FUNCTION_BLOCK FB_System_AFA_600
VAR_INPUT
	Freigabe_auto								: BOOL;
	Freigabe_Deakt_auto							: BOOL;
	Betrieb_Anford_auto							: BOOL;
	Regelung_Modus_auto							: SINT;
	Regelung_Sollw_auto							: REAL;
END_VAR
VAR_OUTPUT
	{attribute 'OPC.UA.DA' := '1'}Steuerung				: ST_System_AFA_Steuerung;		
	{attribute 'OPC.UA.DA' := '1'}Stellwert				: ST_System_AFA_Stellwert;		
	{attribute 'OPC.UA.DA' := '1'}Zustand					: ST_System_AFA_Zustand;	
	{attribute 'OPC.UA.DA' := '1'}Parameter				: ST_System_AFA_Parameter;		
END_VAR
VAR
	Pumpe_600				: FB_PU;
	Pumpe_235				: FB_PU;
	Pumpe_690				: FB_PU_Schuetz;
	Stellventil_605			: FB_SVs;
	Stellventil_235			: FB_SVs;
	Regelventil_600			: FB_RV;
	Regelventil_Ost_640		: FB_RV;
	Regelventil_West_660	: FB_RV;

	Zustandscheck			: FB_System_AFA_Zustandscheck;
	Logik					: FB_System_AFA_Logik;
	Ablaufsteuerung			: FB_System_AFA_Ablaufsteuerung;
	Sollwertscheck			: FB_System_AFA_Sollwertscheck;
	Regelung				: FB_System_AFA_Regelung;
	Stellwertscheck			: FB_System_AFA_Stellwertscheck;
	T_zyklus_ON: TON;
	T_zyklus_OFF: TON;


END_VAR
VAR // added by the converter: edge detectors and wires of the graphical bodies
    _w1 : BOOL;
    _w2 : ANY;
END_VAR

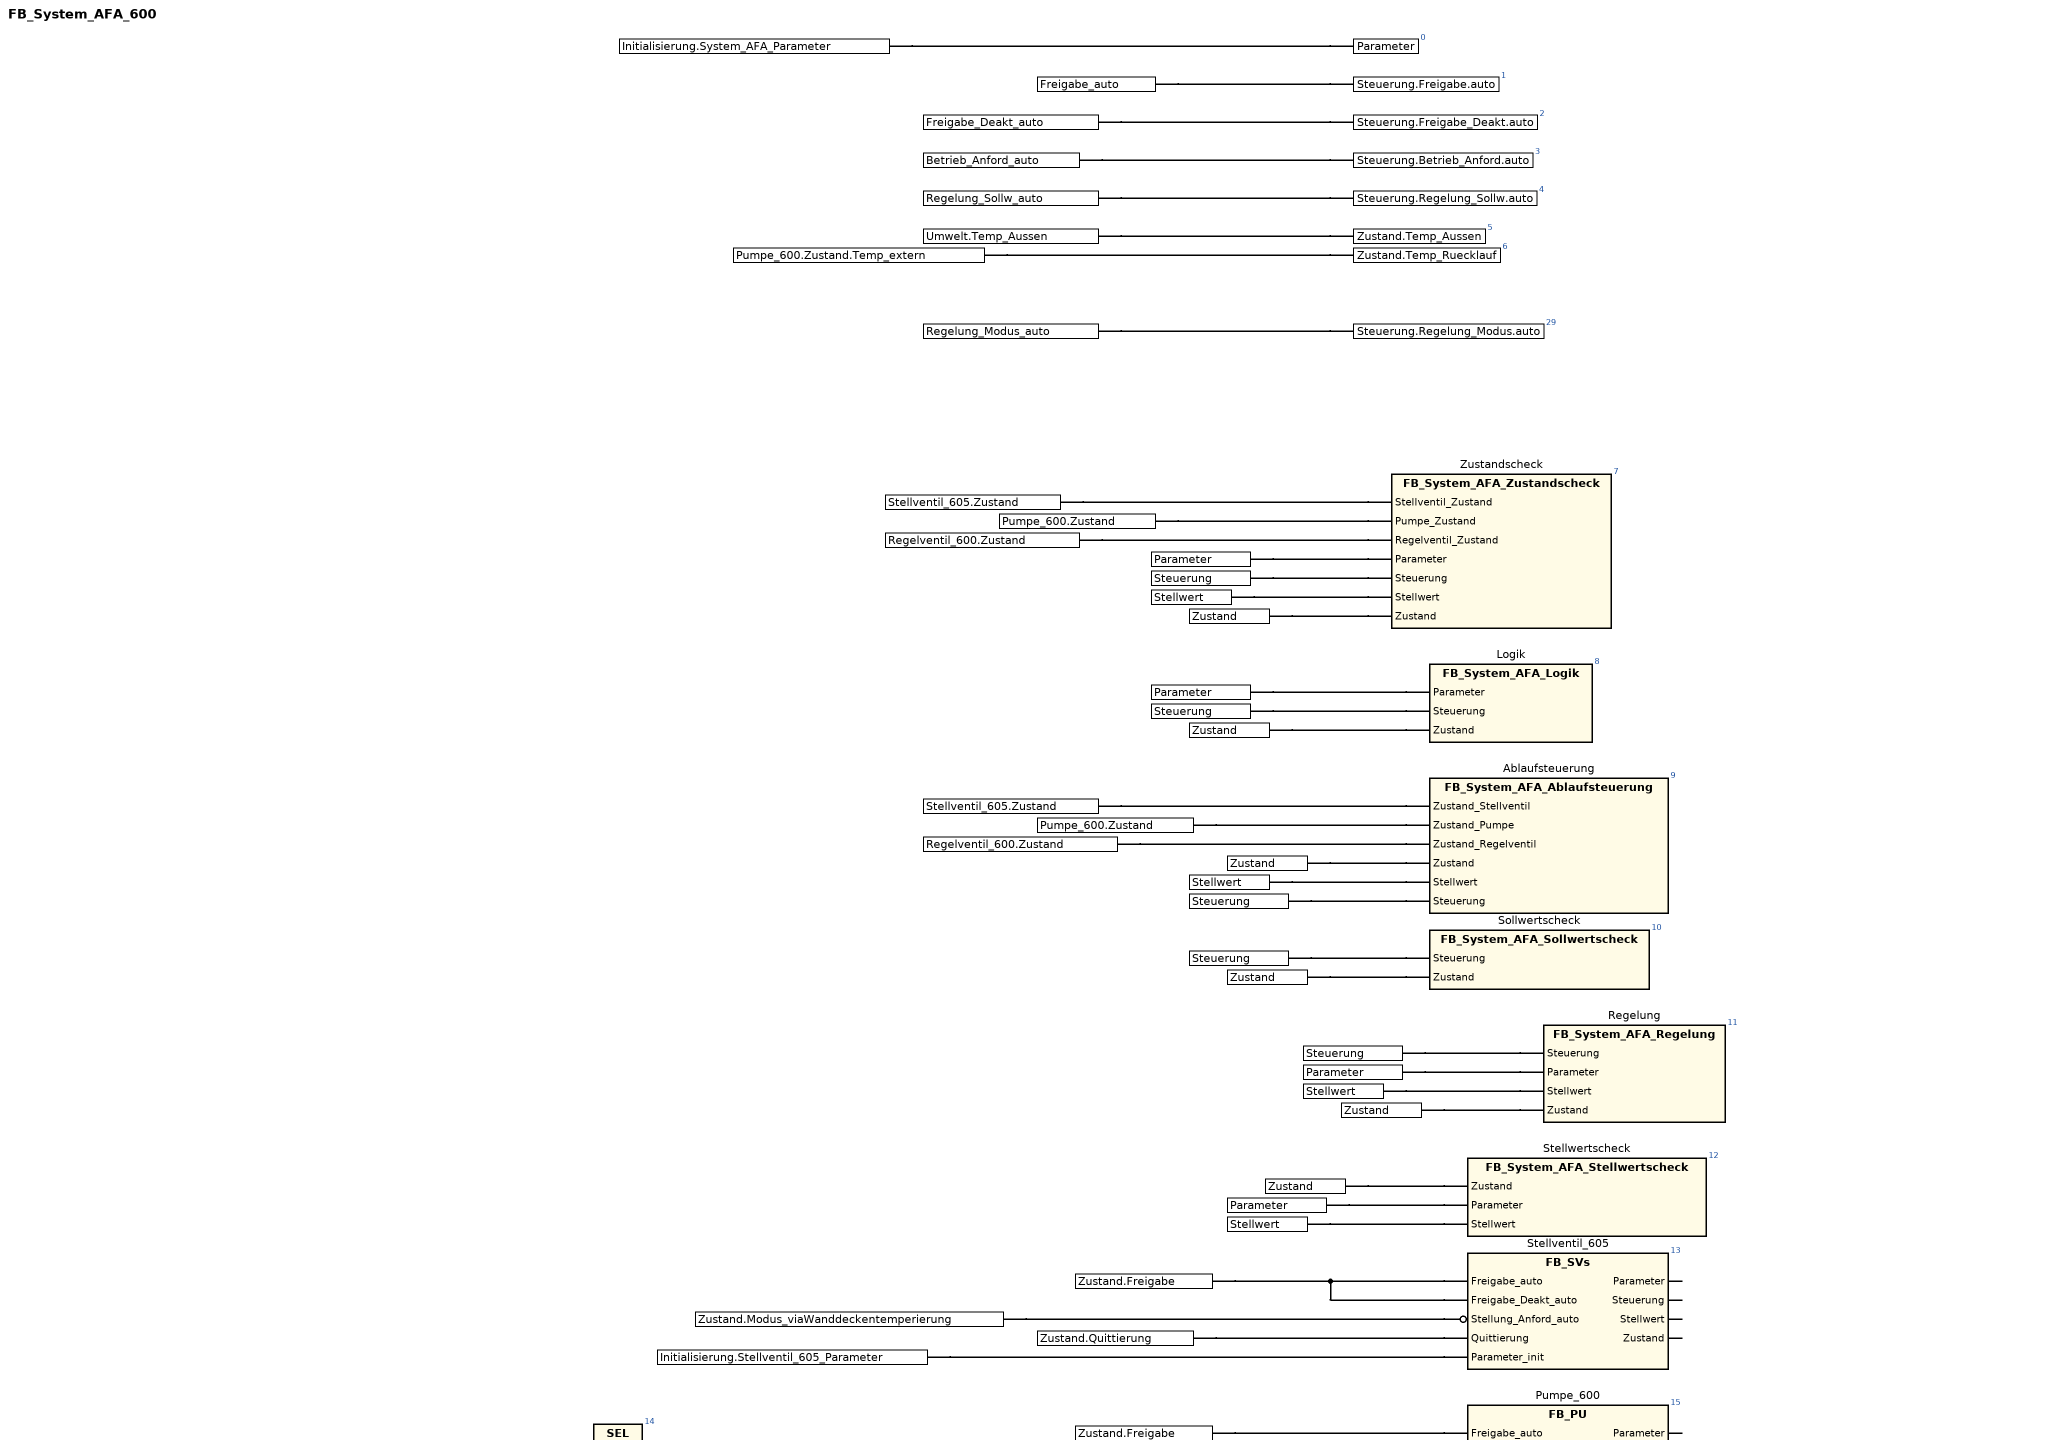
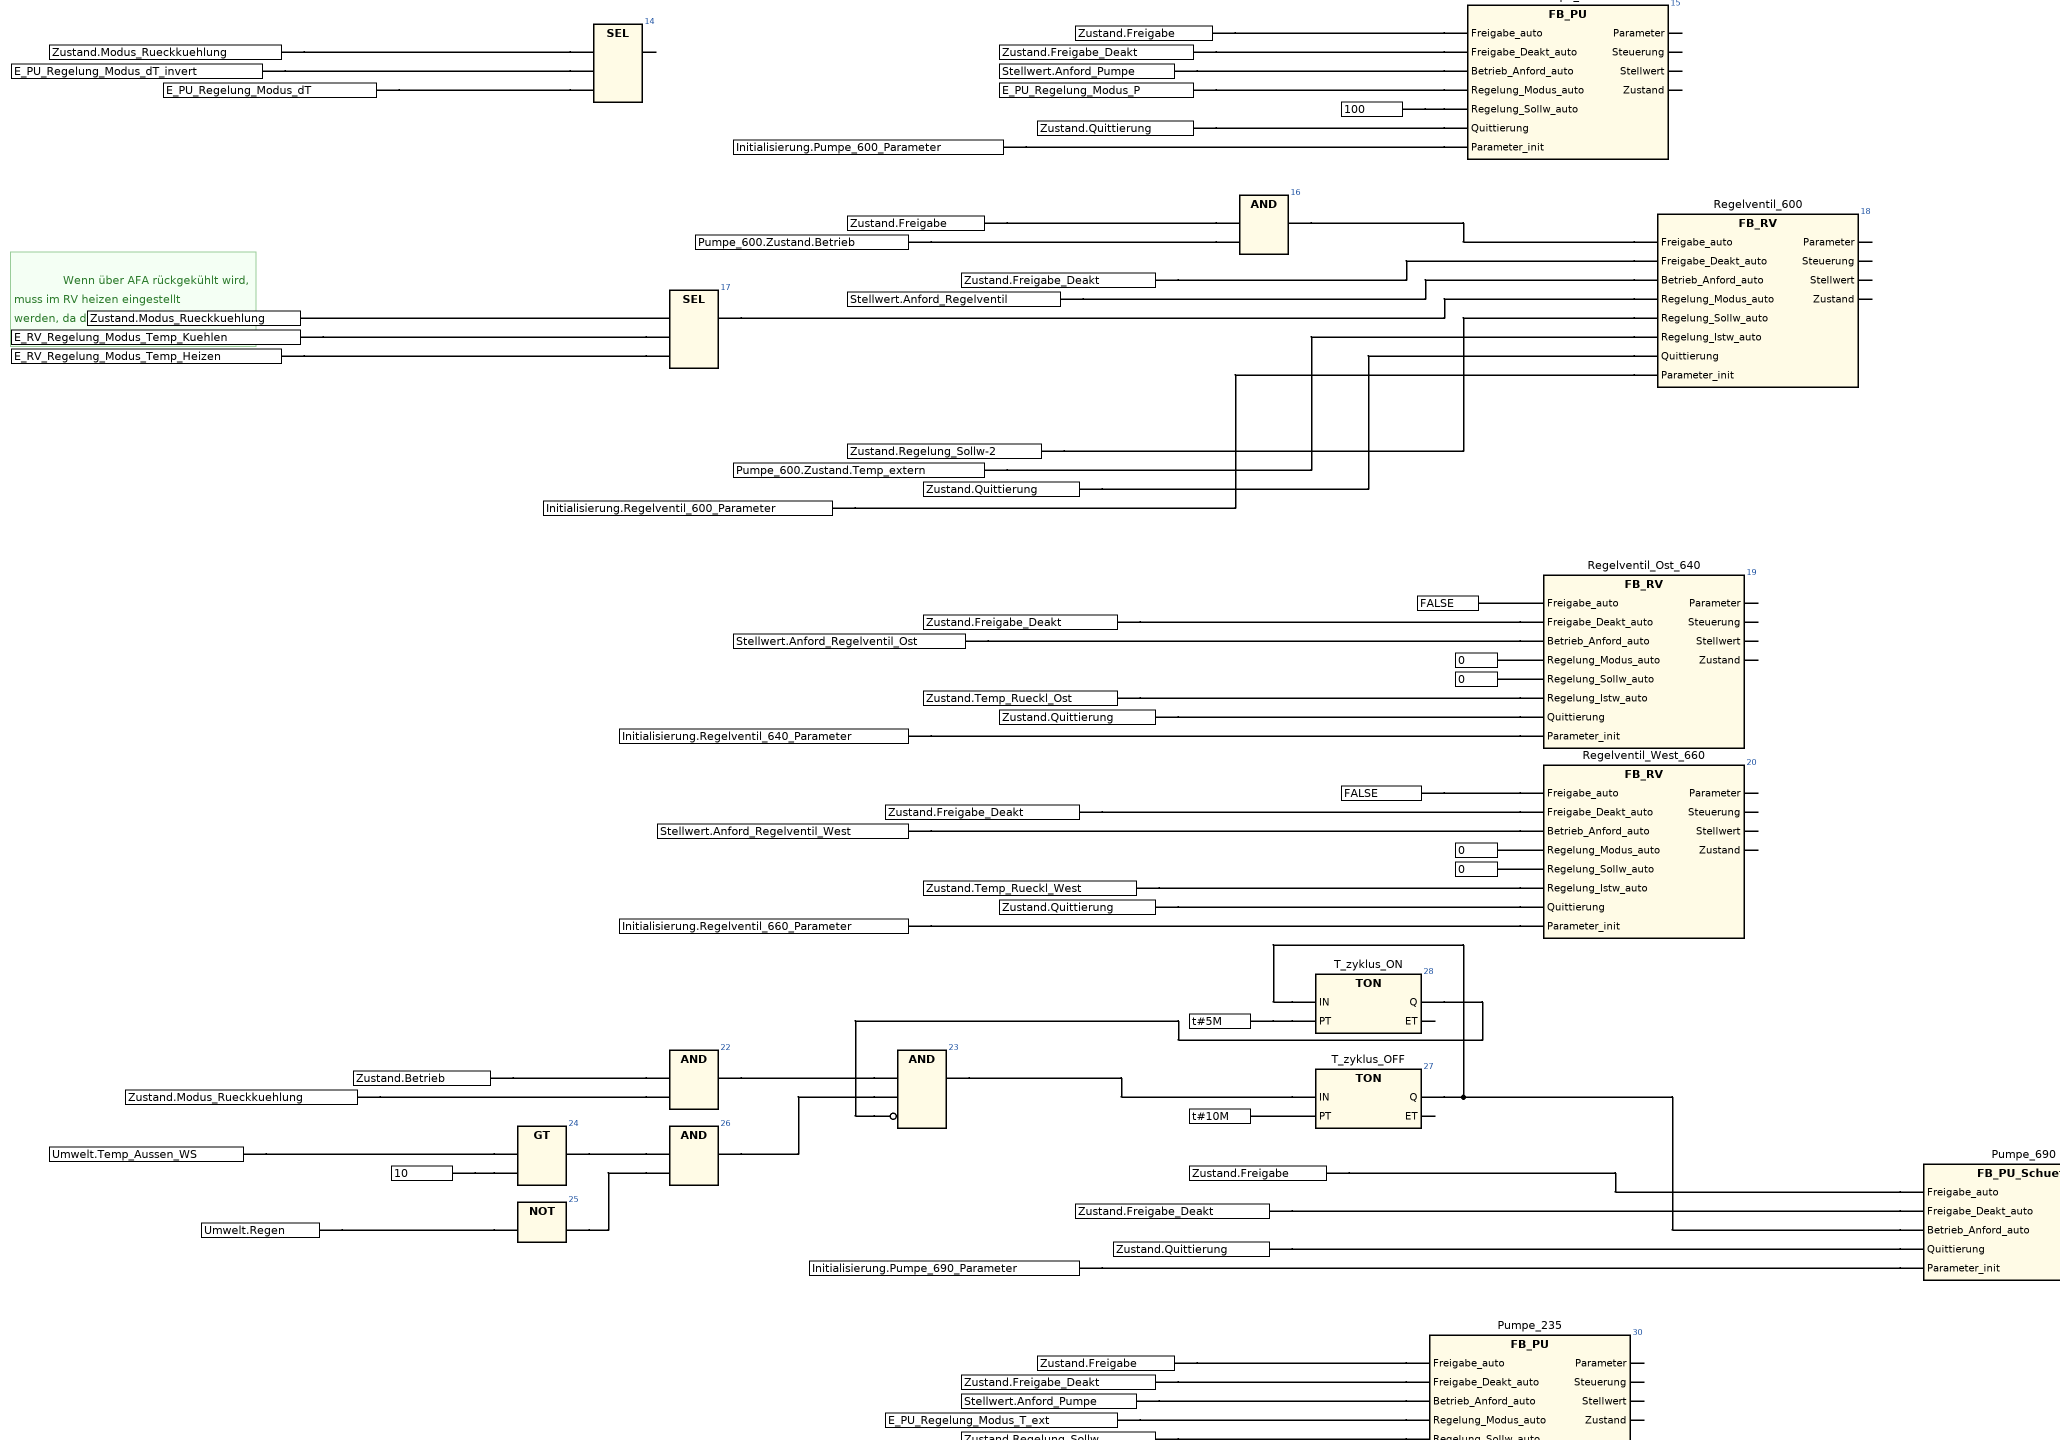
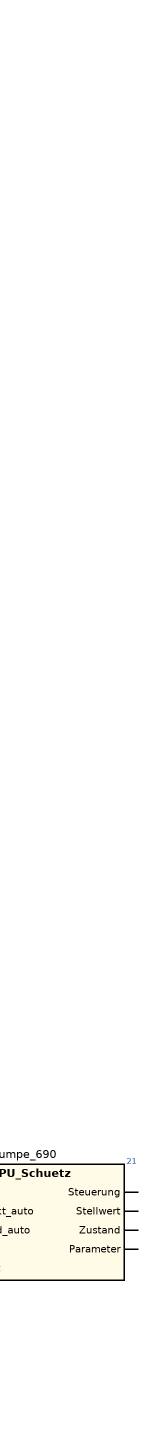
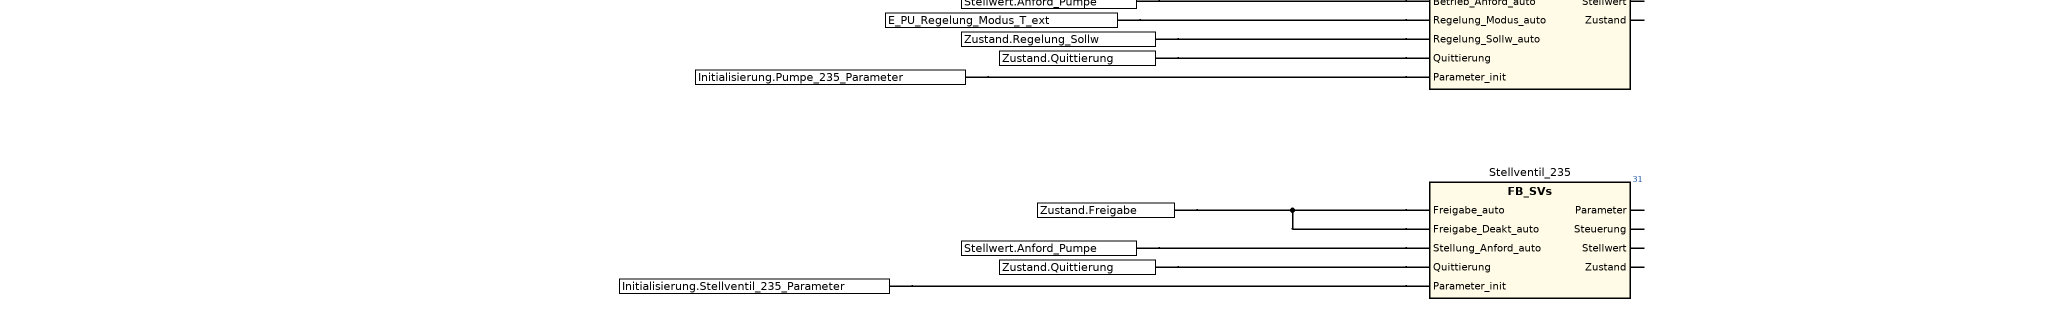
Parameter := Initialisierung.System_AFA_Parameter;
Steuerung.Freigabe.auto := Freigabe_auto;
Steuerung.Freigabe_Deakt.auto := Freigabe_Deakt_auto;
Steuerung.Betrieb_Anford.auto := Betrieb_Anford_auto;
Steuerung.Regelung_Sollw.auto := Regelung_Sollw_auto;
Zustand.Temp_Aussen := Umwelt.Temp_Aussen;
Zustand.Temp_Ruecklauf := Pumpe_600.Zustand.Temp_extern;
Zustandscheck(
    Stellventil_Zustand := Stellventil_605.Zustand,
    Pumpe_Zustand := Pumpe_600.Zustand,
    Regelventil_Zustand := Regelventil_600.Zustand,
    Parameter := Parameter,
    Steuerung := Steuerung,
    Stellwert := Stellwert,
    Zustand := Zustand); // FB_System_AFA_Zustandscheck
Logik(Parameter := Parameter, Steuerung := Steuerung, Zustand := Zustand); // FB_System_AFA_Logik
Ablaufsteuerung(
    Zustand_Stellventil := Stellventil_605.Zustand,
    Zustand_Pumpe := Pumpe_600.Zustand,
    Zustand_Regelventil := Regelventil_600.Zustand,
    Zustand := Zustand,
    Stellwert := Stellwert,
    Steuerung := Steuerung); // FB_System_AFA_Ablaufsteuerung
Sollwertscheck(Steuerung := Steuerung, Zustand := Zustand); // FB_System_AFA_Sollwertscheck
Regelung(Steuerung := Steuerung, Parameter := Parameter, Stellwert := Stellwert, Zustand := Zustand); // FB_System_AFA_Regelung
Stellwertscheck(Zustand := Zustand, Parameter := Parameter, Stellwert := Stellwert); // FB_System_AFA_Stellwertscheck
Stellventil_605(
    Freigabe_auto := Zustand.Freigabe,
    Freigabe_Deakt_auto := Zustand.Freigabe,
    Stellung_Anford_auto := NOT Zustand.Modus_viaWanddeckentemperierung,
    Quittierung := Zustand.Quittierung,
    Parameter_init := Initialisierung.Stellventil_605_Parameter); // FB_SVs
(* SEL(Zustand.Modus_Rueckkuehlung, E_PU_Regelung_Modus_dT_invert, E_PU_Regelung_Modus_dT); result not used *)
Pumpe_600(
    Freigabe_auto := Zustand.Freigabe,
    Freigabe_Deakt_auto := Zustand.Freigabe_Deakt,
    Betrieb_Anford_auto := Stellwert.Anford_Pumpe,
    Regelung_Modus_auto := E_PU_Regelung_Modus_P,
    Regelung_Sollw_auto := 100,
    Quittierung := Zustand.Quittierung,
    Parameter_init := Initialisierung.Pumpe_600_Parameter); // FB_PU
// 							Wenn über AFA rückgekühlt wird,
// muss im RV heizen eingestellt
// werden, da die AFA "beheizt" wird
//
Regelventil_600(
    Freigabe_auto := Zustand.Freigabe AND Pumpe_600.Zustand.Betrieb,
    Freigabe_Deakt_auto := Zustand.Freigabe_Deakt,
    Betrieb_Anford_auto := Stellwert.Anford_Regelventil,
    Regelung_Modus_auto := SEL(Zustand.Modus_Rueckkuehlung, E_RV_Regelung_Modus_Temp_Kuehlen, E_RV_Regelung_Modus_Temp_Heizen),
    Regelung_Sollw_auto := Zustand.Regelung_Sollw-2,
    Regelung_Istw_auto := Pumpe_600.Zustand.Temp_extern,
    Quittierung := Zustand.Quittierung,
    Parameter_init := Initialisierung.Regelventil_600_Parameter); // FB_RV
Regelventil_Ost_640(
    Freigabe_auto := FALSE,
    Freigabe_Deakt_auto := Zustand.Freigabe_Deakt,
    Betrieb_Anford_auto := Stellwert.Anford_Regelventil_Ost,
    Regelung_Modus_auto := 0,
    Regelung_Sollw_auto := 0,
    Regelung_Istw_auto := Zustand.Temp_Rueckl_Ost,
    Quittierung := Zustand.Quittierung,
    Parameter_init := Initialisierung.Regelventil_640_Parameter); // FB_RV
Regelventil_West_660(
    Freigabe_auto := FALSE,
    Freigabe_Deakt_auto := Zustand.Freigabe_Deakt,
    Betrieb_Anford_auto := Stellwert.Anford_Regelventil_West,
    Regelung_Modus_auto := 0,
    Regelung_Sollw_auto := 0,
    Regelung_Istw_auto := Zustand.Temp_Rueckl_West,
    Quittierung := Zustand.Quittierung,
    Parameter_init := Initialisierung.Regelventil_660_Parameter); // FB_RV
Pumpe_690(
    Freigabe_auto := Zustand.Freigabe,
    Freigabe_Deakt_auto := Zustand.Freigabe_Deakt,
    Betrieb_Anford_auto := T_zyklus_OFF.Q,
    Quittierung := Zustand.Quittierung,
    Parameter_init := Initialisierung.Pumpe_690_Parameter); // FB_PU_Schuetz
_w2 := (Zustand.Betrieb AND Zustand.Modus_Rueckkuehlung) AND _w1 AND NOT T_zyklus_ON.Q;
_w1 := Umwelt.Temp_Aussen_WS > 10 AND NOT Umwelt.Regen;
T_zyklus_OFF(IN := _w2, PT := t#10M); // TON
T_zyklus_ON(IN := T_zyklus_OFF.Q, PT := t#5M); // TON
Steuerung.Regelung_Modus.auto := Regelung_Modus_auto;
Pumpe_235(
    Freigabe_auto := Zustand.Freigabe,
    Freigabe_Deakt_auto := Zustand.Freigabe_Deakt,
    Betrieb_Anford_auto := Stellwert.Anford_Pumpe,
    Regelung_Modus_auto := E_PU_Regelung_Modus_T_ext,
    Regelung_Sollw_auto := Zustand.Regelung_Sollw,
    Quittierung := Zustand.Quittierung,
    Parameter_init := Initialisierung.Pumpe_235_Parameter); // FB_PU
Stellventil_235(
    Freigabe_auto := Zustand.Freigabe,
    Freigabe_Deakt_auto := Zustand.Freigabe,
    Stellung_Anford_auto := Stellwert.Anford_Pumpe,
    Quittierung := Zustand.Quittierung,
    Parameter_init := Initialisierung.Stellventil_235_Parameter); // FB_SVs

END_FUNCTION_BLOCK

(* stored: Version 1.1.0.1, ProductVersion 3.1.4024.9
   POU FB_System_AFA_600: Id {1ef46571-5e93-4d88-98f8-b2ca23d6f556}, SpecialFunc None *)
